PROGRAM MAIN
VAR
	dataTests : TestDataContext;
	sandbox : SandboxContext;
END_VAR

dataTests.ProbeRun();
sandbox.Run();

END_PROGRAM

(* stored: Version 1.1.0.1, ProductVersion 3.1.4024.9
   POU MAIN: Id {0f34ba18-e40b-0caf-2a51-227dede86d56}, SpecialFunc None *)
